(*********************************** G.D S.p.A. - Technical Department ***********************************
============= PROGRAM INFO ============
FOLDER:             TBD
MACHINES INVOLVED:  TBD 

============= DESCRIPTION =============
csp machine declaration

============= REVISIONS ===============
Date		Version	 	Author      	Description             
----------	-------		------------  	--------------------------------------------
2019/04/05 	0000.00	 	M.Grasso		Creation of the PRG

**********************************************************************************************************)
(*$R process_ref := prc; $*)
PROGRAM csp_case_tr_accU_os
VAR
	
	prc:											process;
	prc_path:										STRING;
	
END_VAR

_read_var_input();

_object_manager();

IF NOT objects_running()
THEN
	RETURN;	
END_IF

_read_process_image();

_mode_manager();

_set_runtime_properties();

(********************************* BODY *********************************)
(************************************************************************)

_handle_messages();

_write_output();

ACTION _handle_messages:
;
END_ACTION

ACTION _handle_process_test:
;
END_ACTION

ACTION _mode_manager:
IF process_mode_req_is_pending(prc)
THEN
    process_apply_mode_req_first_step(prc);
    CASE process_get_mode(prc) OF
        MODE_TO_ABSENT:
			;
        MODE_TO_INACTIVE:
			;
        MODE_TO_TEST:
			;
        MODE_TO_OPERATIONAL:
			;
    END_CASE
    process_apply_mode_req_second_step(prc);
END_IF
END_ACTION

ACTION _object_manager:
IF objects_initialization()
THEN
	sub_process_init(
		object_name					:= 'csp_case_tr_accU_os.prc', 
		process						:= csp_case_topRail_accU.prc, 
		CONVERSION_this				:= prc);
		
	prc_path 						:= process_get_path(prc);
END_IF

IF objects_running()
THEN
	process_cycle(prc);
END_IF
END_ACTION

ACTION _read_process_image:
;
END_ACTION

ACTION _read_var_input:
;
END_ACTION

ACTION _set_runtime_properties:
;
END_ACTION

ACTION _write_output:
;
END_ACTION

END_PROGRAM

(* stored: Version 1.1.0.1, ProductVersion 3.1.4022.12
   POU csp_case_tr_accU_os: Id {78a7a66d-3b41-459c-a275-945343af8335}, SpecialFunc None
   Action _handle_messages: Id {fc9c4709-cee3-4321-8fcf-bb60883ff3ce}
   Action _handle_process_test: Id {2373846f-5e2e-4e66-ab5f-0ed2bd4285f0}
   Action _mode_manager: Id {f48e3f89-2002-4977-8909-c38042fcca52}
   Action _object_manager: Id {38d501e2-07f7-4a07-ac91-3ce73b14b1c2}
   Action _read_process_image: Id {8ffaf1c7-505f-4523-91af-d04bbe091b18}
   Action _read_var_input: Id {586c0f61-104b-494c-a8bc-11d1c3048df3}
   Action _set_runtime_properties: Id {f9de6bdf-a265-487b-a8be-9f7e2ae56ad8}
   Action _write_output: Id {83f4aa92-3799-4563-b652-024dc76cd99d} *)
